// TIA Portal V16 export
// export: Created 2022-09-01T14:29:23.3813715Z, ExportSetting WithDefaults, DisplayName Totally Integrated Automation Portal, DisplayVersion V16, DisplayName TIA Portal Version Control Interface, DisplayVersion V16, DisplayName TIA Portal Openness, DisplayVersion V16, DisplayName STEP 7 Professional, DisplayVersion V16, DisplayName STEP 7 Safety, DisplayVersion V16, DisplayName WinCC Advanced, DisplayVersion V16
FUNCTION "Reinício_Ciclo" : Void   // FC19, LAD
{ S7_Optimized_Access := 'TRUE' }
VERSION : 0.1
// stored: AutoNumber true, IsIECCheckEnabled false, SetENOAutomatically false, UDAEnableTagReadback false
   VAR_TEMP   // added for the SCL form of the ladder/FBD networks
      _w1 : Bool;
   END_VAR
BEGIN

REGION Network 1: Ativa etapa 1 e faz reset às restantes do ciclo de tratamento
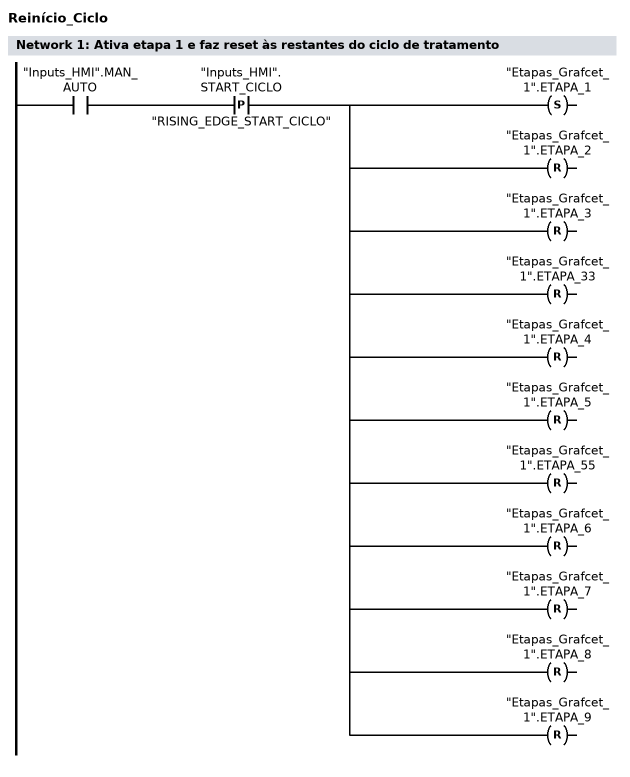
   RUNG wire#powerrail
      Contact( "Inputs_HMI".MAN_AUTO )
      P_Contact(operand := "Inputs_HMI".START_CICLO, bit := "RISING_EDGE_START_CICLO")
      wire#w1
      S_Coil( "Etapas_Grafcet_1".ETAPA_1 )
   END_RUNG
   RUNG wire#w1
      R_Coil( "Etapas_Grafcet_1".ETAPA_2 )
   END_RUNG
   RUNG wire#w1
      R_Coil( "Etapas_Grafcet_1".ETAPA_3 )
   END_RUNG
   RUNG wire#w1
      R_Coil( "Etapas_Grafcet_1".ETAPA_33 )
   END_RUNG
   RUNG wire#w1
      R_Coil( "Etapas_Grafcet_1".ETAPA_4 )
   END_RUNG
   RUNG wire#w1
      R_Coil( "Etapas_Grafcet_1".ETAPA_5 )
   END_RUNG
   RUNG wire#w1
      R_Coil( "Etapas_Grafcet_1".ETAPA_55 )
   END_RUNG
   RUNG wire#w1
      R_Coil( "Etapas_Grafcet_1".ETAPA_6 )
   END_RUNG
   RUNG wire#w1
      R_Coil( "Etapas_Grafcet_1".ETAPA_7 )
   END_RUNG
   RUNG wire#w1
      R_Coil( "Etapas_Grafcet_1".ETAPA_8 )
   END_RUNG
   RUNG wire#w1
      R_Coil( "Etapas_Grafcet_1".ETAPA_9 )
   END_RUNG
   // the same network as SCL:
   #_w1 := "Inputs_HMI".MAN_AUTO AND "Inputs_HMI".START_CICLO AND NOT "RISING_EDGE_START_CICLO";   // rising edge of "Inputs_HMI".START_CICLO
   "RISING_EDGE_START_CICLO" := "Inputs_HMI".START_CICLO;
   IF #_w1 THEN
       "Etapas_Grafcet_1".ETAPA_1 := TRUE;
       "Etapas_Grafcet_1".ETAPA_2 := FALSE;
       "Etapas_Grafcet_1".ETAPA_3 := FALSE;
       "Etapas_Grafcet_1".ETAPA_33 := FALSE;
       "Etapas_Grafcet_1".ETAPA_4 := FALSE;
       "Etapas_Grafcet_1".ETAPA_5 := FALSE;
       "Etapas_Grafcet_1".ETAPA_55 := FALSE;
       "Etapas_Grafcet_1".ETAPA_6 := FALSE;
       "Etapas_Grafcet_1".ETAPA_7 := FALSE;
       "Etapas_Grafcet_1".ETAPA_8 := FALSE;
       "Etapas_Grafcet_1".ETAPA_9 := FALSE;
   END_IF;
END_REGION
END_FUNCTION
